TYPE TcaTrolleyRef :
STRUCT
	Sensor AT%I* : BOOL;	
END_STRUCT
END_TYPE

(* stored: Version 1.1.0.1
   DUT TcaTrolleyRef: Id {a334b748-4b7a-4e04-8e56-b4a81f775b6c} *)
